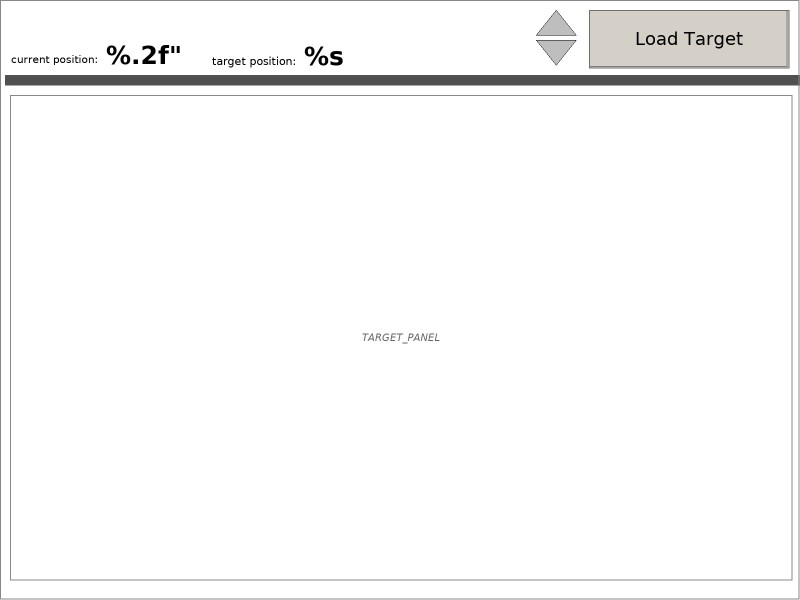
VISUALIZATION MAIN_DASHBOARD  // 800x600
    Rectangle (0,0 810x600)
    Button (589,10 200x58), "Unload Target", colour toggle: GV_HMI.colortoggle[6]
        tap GV_HMI.colortoggle[6]
        OnMouseDown: execute { HMI.bTgtLoaded := FALSE; GV_LIFT.MTP_ALLOWED := FALSE; }
    Rectangle (5,75 795x10)
    Rectangle (12,50 89x19), "current position:"
    Rectangle (103,40 135x30), "%.2f"", text variable: GV_LIFT.CURRENT_POSITION
    Rectangle (208,52 91x19), "target position:"
    Rectangle (301,39 132x34), "%s", text variable: HMI.DisplayTgtPos, invisible if: GV_LIFT.MTP_ALLOWED <>1
    Button (589,10 200x58), "Load Target", colour toggle: GV_HMI.colortoggle[6], invisible if: HMI.bUnload <> 0, input disabled if: HMI.bLoadOK<>1
        tap GV_HMI.colortoggle[6]
        OnMouseDown: execute {
            GV_LIFT.TARGET_POSITION := XML.savedvalues.savedpos[GV_HMI.RowSelect].target;
            GV_HMI.RowSelected := GV_HMI.RowSelect;
            HMI.bTgtLoaded := TRUE;
            GV_LIFT.MTP_ALLOWED := TRUE;
            GV_LIFT.JUST_RAN := FALSE;
        }
    TabControl (10,95 782x485)
        shows TARGET_PANEL()
        shows SAFETY_PANEL()
        shows Visualization_2()
        shows Visualization_2()
        shows Visualization_2()
        [0]: TabTitle=Target Positions
        [1]: TabTitle=Safety Status Panel
    Polygon (536,35) (556,10) (576,35) (576,35) (536,35), colour variable: HMI_Up_Arrow_Indicator.dwUpArrow
    Polygon (536,40) (556,65) (576,40) (576,40) (536,40), colour variable: HMI_Down_Arrow_Indicator.dwDownArrow
END_VISUALIZATION

(* stored: Version 1.1.0.1, ProductVersion 3.1.4022.12
   Visu MAIN_DASHBOARD: Id {c482051d-8314-45a1-96c5-8e033d44a6f5} *)
